/// Control cabinet IOs
TYPE ST_ControlCabinetIO :
STRUCT
	stIn	AT%I* : ST_ControlCabinetIn;
	stOut	AT%Q* : ST_ControlCabinetOut;
END_STRUCT
END_TYPE

(* stored: Version 1.1.0.1, ProductVersion 3.1.4024.12
   DUT ST_ControlCabinetIO: Id {9ba3c62d-3fc3-42a8-9a71-d9fca44b04bc} *)
